FUNCTION TEN : LREAL
VAR_INPUT
	dd,mm,ss: LREAL;
END_VAR
VAR
END_VAR

TEN := dd + (mm/60.0) + (ss/3600.0);

END_FUNCTION

(* stored: Version 1.1.0.1, ProductVersion 3.1.4024.0
   POU TEN: Id {48a4167d-326b-4179-a49a-d85a103bff69}, SpecialFunc None *)
